ABB RobotStudio station: saddlewelding_2dofpositioner.rspag

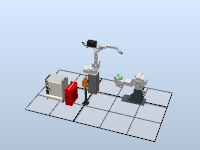
--- station ---
Station FInal3_1520_2dof (saved by RobotStudio 7.0.8743.626)
Controller Final3_1520_2dof, task T_ROB1: task frame (RAPID world) sits at (0, 0, 900) mm in the station
Controller Final3_1520_2dof
  mechanical unit ROB_1: IRB1520ID_4_150__02, 6 joints, base frame (0, 0, 0) mm
  mechanical unit STN1: IRBP_A250_D1000_M2009_REV1_01, 2 joints, base frame (0, 0, 0) mm
Layout (positions relative to the parent item):
  - IRB1520ID_4_150__02 [mechanism, from Robots\IRB1520ID_4_150_G_02.rslib] at (0, 0, 900) mm; joint values [0, 0, 0, 0, 0.5236, 0] (rad or m)
  - base900 [part, from Dissertation\base900.rslib]
  - IRBP_A250_D1000_M2009_REV1_01 [mechanism] at (1025, 0, 0) mm; joint values [0, 0] (rad or m)
      links: Base, Link1, Link2
  - Binzel_ID_22 [mechanism, from Tools\Binzel_ID_22.rslib] at (1056.21, 0, 2043) mm, rotated rx 180 ry 60 rz 180 deg
  - saddle_simple_tpipe [part] at (1025, 0, 940) mm, rotated rx 90 ry 0 rz 180 deg
  - Fronius_VR1500 [part, from Equipment\Fronius_VR1500.rslib] at (-224.71, 27.64, 723.67) mm
  - IRC5_Singel-Cabinet [part, from Equipment\IRC5_Singel-Cabinet.rslib] at (-1184.73, -1000, 100) mm, rotated rx 90 ry 0 rz 0 deg
  - Fronius_TPS4000_rev0 [part, from Equipment\Fronius_TPS4000.rslib] at (-575.52, -881.82, 0) mm, rotated rx 0 ry 0 rz 180 deg
  - torch_cleaner_binzel [graphiccomponentgroup, from Equipment\Torch Cleaner Binzel.rslib] at (0, -815.14, 0) mm
    - Body 1 [part, from Equipment\Torch Cleaner Binzel.rslib]
    - Body 2 [part, from Equipment\Torch Cleaner Binzel.rslib]
    - Body 3 [part, from Equipment\Torch Cleaner Binzel.rslib]
    - Body 4 [part, from Equipment\Torch Cleaner Binzel.rslib]
    - Body 5 [part, from Equipment\Torch Cleaner Binzel.rslib]
    - Body 6 [part, from Equipment\Torch Cleaner Binzel.rslib]
    - Body 7 [part, from Equipment\Torch Cleaner Binzel.rslib]
    - Body 8 [part, from Equipment\Torch Cleaner Binzel.rslib]
    - Body 9 [part, from Equipment\Torch Cleaner Binzel.rslib]
    - Body 10 [part, from Equipment\Torch Cleaner Binzel.rslib]
    - Body 11 [part, from Equipment\Torch Cleaner Binzel.rslib]
    - Body 12 [part, from Equipment\Torch Cleaner Binzel.rslib]
Attachment: Binzel_ID_22 is attached to IRB1520ID_4_150__02 / Link6
Attachment: saddle_simple_tpipe is attached to IRBP_A250_D1000_M2009_REV1_01 / Link2
Attachment: Fronius_VR1500 is attached to IRB1520ID_4_150__02 / Link3

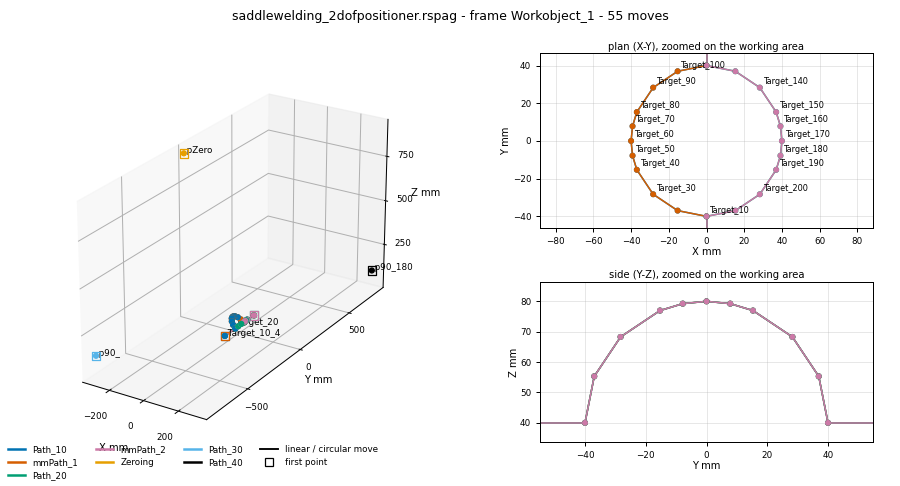
[picture p0: tool path of saddlewelding_2dofpositioner.rspag in frame Workobject_1, 55 of 55 moves have a stored position in this frame; points joined in program order, loops and branches not executed]
--- Backups/Final3_1520_2dof/RAPID/TASK1/PROGMOD/CalibData.mod ---
MODULE CalibData
	PERS tooldata tWeldGun:=[TRUE,[[49.841566361,0,372.194826196],[0.981627183,0,0.190808995,0]],[2,[0,0,100],[0,1,0,0],0,0,0]];
	TASK PERS wobjdata Workobject_1:=[FALSE,FALSE,"STN1",[[0,0,0],[1,0,0,0]],[[0,0,0],[1,0,0,0]]];
ENDMODULE

--- Backups/Final3_1520_2dof/RAPID/TASK1/PROGMOD/Module1.mod ---
MODULE Module1
	CONST robtarget Target_10_4:=[[0,-140,40],[0.653281482,-0.653281483,-0.27059805,-0.27059805],[0,0,0,0],[9E+09,9E+09,9E+09,9E+09,9E+09,9E+09]];
	CONST robtarget Target_10:=[[0,-40,40],[0.653281482,-0.653281483,-0.27059805,-0.27059805],[0,0,0,0],[9E+09,9E+09,9E+09,9E+09,9E+09,9E+09]];
	CONST robtarget Target_20:=[[-15.307337295,-36.9551813,55.307337295],[0.552498444,-0.741273461,-0.232815701,-0.301754825],[0,0,0,0],[9E+09,9E+09,9E+09,9E+09,9E+09,9E+09]];
	CONST robtarget Target_30:=[[-28.284271247,-28.284271247,68.284271247],[0.424708201,-0.820473238,-0.175919897,-0.339851143],[0,0,0,0],[9E+09,9E+09,9E+09,9E+09,9E+09,9E+09]];
	CONST robtarget Target_40:=[[-36.9551813,-15.307337295,76.9551813],[0.245447259,-0.877471606,-0.091255347,-0.401835396],[0,0,0,0],[9E+09,9E+09,9E+09,9E+09,9E+09,9E+09]];
	CONST robtarget Target_50:=[[-39.231411216,-7.803612881,79.231411216],[0.126767777,-0.911559828,-0.051100945,-0.387785125],[0,0,0,0],[9E+09,9E+09,9E+09,9E+09,9E+09,9E+09]];
	CONST robtarget Target_60:=[[-40,0,80],[0,0.923879533,0,0.382683432],[0,0,0,0],[9E+09,9E+09,9E+09,9E+09,9E+09,9E+09]];
	CONST robtarget Target_70:=[[-39.231411216,7.803612881,79.231411216],[0.126767777,0.911559828,-0.051100945,0.387785125],[0,0,0,0],[9E+09,9E+09,9E+09,9E+09,9E+09,9E+09]];
	CONST robtarget Target_80:=[[-36.9551813,15.307337295,76.9551813],[0.245447259,0.877471606,-0.091255347,0.401835396],[0,0,0,0],[9E+09,9E+09,9E+09,9E+09,9E+09,9E+09]];
	CONST robtarget Target_90:=[[-28.284271247,28.284271247,68.284271247],[0.424708201,0.820473238,-0.175919897,0.339851143],[0,0,0,0],[9E+09,9E+09,9E+09,9E+09,9E+09,9E+09]];
	CONST robtarget Target_100:=[[-15.307337295,36.9551813,55.307337295],[0.552498444,0.741273461,-0.232815702,0.301754825],[0,0,0,0],[9E+09,9E+09,9E+09,9E+09,9E+09,9E+09]];
	CONST robtarget Target_110:=[[0,40,40],[0.653281482,0.653281483,-0.27059805,0.27059805],[0,0,0,0],[9E+09,9E+09,9E+09,9E+09,9E+09,9E+09]];
	CONST robtarget Target_110_3:=[[0,140,40],[0.653281482,0.653281483,-0.27059805,0.27059805],[0,0,0,0],[9E+09,9E+09,9E+09,9E+09,9E+09,9E+09]];
	CONST robtarget pTarget_1:=[[0,-140,40],[0.653281482,-0.653281483,-0.27059805,-0.27059805],[-1,0,-1,0],[9E+09,-89.999998314,-0.000000734,9E+09,9E+09,9E+09]];
	CONST robtarget pTarget_2:=[[0,-40,40],[0.653281482,-0.653281483,-0.27059805,-0.27059805],[-1,0,-1,0],[9E+09,-89.802410692,4.557172082,9E+09,9E+09,9E+09]];
	CONST robtarget pTarget_3:=[[-15.307337295,-36.9551813,55.307337295],[0.552498444,-0.741273461,-0.232815701,-0.301754825],[-1,0,-1,0],[9E+09,-76.295977766,18.279214138,9E+09,9E+09,9E+09]];
	CONST robtarget pTarget_4:=[[-28.284271247,-28.284271247,68.284271247],[0.424708201,-0.820473238,-0.175919897,-0.339851143],[-1,0,-1,0],[9E+09,-61.411118651,37.565448127,9E+09,9E+09,9E+09]];
	CONST robtarget pTarget_5:=[[-36.9551813,-15.307337295,76.9551813],[0.245447259,-0.877471606,-0.091255347,-0.401835396],[-1,0,-2,0],[9E+09,-47.380570194,71.170137619,9E+09,9E+09,9E+09]];
	CONST robtarget pTarget_6:=[[-39.231411216,-7.803612881,79.231411216],[0.126767777,-0.911559828,-0.051100945,-0.387785125],[-1,0,-2,0],[9E+09,-36.088107809,97.239437874,9E+09,9E+09,9E+09]];
	CONST robtarget pTarget_7:=[[-40,0,80],[0,0.923879533,0,0.382683432],[-1,0,-2,0],[9E+09,-31.001963049,129.358833622,9E+09,9E+09,9E+09]];
	CONST robtarget pTarget_8:=[[-39.231411216,7.803612881,79.231411216],[0.126767777,0.911559828,-0.051100945,0.387785125],[-1,0,-2,0],[9E+09,-36.088107791,152.02186895,9E+09,9E+09,9E+09]];
	CONST robtarget pTarget_9:=[[-36.9551813,15.307337295,76.9551813],[0.245447259,0.877471606,-0.091255347,0.401835396],[-1,0,-2,0],[9E+09,-47.380570194,163.079129504,9E+09,9E+09,9E+09]];
	CONST robtarget pTarget_10:=[[-28.284271247,28.284271247,68.284271247],[0.424708201,0.820473238,-0.175919897,0.339851143],[-1,0,-2,0],[9E+09,-61.411118652,186.252573581,9E+09,9E+09,9E+09]];
	CONST robtarget pTarget_11:=[[-15.307337295,36.9551813,55.307337295],[0.552498444,0.741273461,-0.232815702,0.301754825],[-1,0,-2,0],[9E+09,-76.29597773,198.192760331,9E+09,9E+09,9E+09]];
	CONST robtarget pTarget_12:=[[0,40,40],[0.653281482,0.653281483,-0.27059805,0.27059805],[-1,0,-2,0],[9E+09,-89.802410695,207.373271387,9E+09,9E+09,9E+09]];
	CONST robtarget pTarget_13:=[[0,140,40],[0.653281482,0.653281483,-0.27059805,0.27059805],[-1,0,-2,0],[9E+09,-89.999998314,199.574847217,9E+09,9E+09,9E+09]];
	CONST robtarget Target_120_2:=[[0,140,40],[0.27059805,0.27059805,-0.653281483,0.653281482],[0,0,0,0],[9E+09,9E+09,9E+09,9E+09,9E+09,9E+09]];
	CONST robtarget Target_120:=[[0,40,40],[0.27059805,0.27059805,-0.653281483,0.653281482],[0,0,0,0],[9E+09,9E+09,9E+09,9E+09,9E+09,9E+09]];
	CONST robtarget Target_130:=[[15.307337295,36.9551813,55.307337295],[0.301754825,0.232815701,-0.741273461,0.552498444],[0,0,0,0],[9E+09,9E+09,9E+09,9E+09,9E+09,9E+09]];
	CONST robtarget Target_140:=[[28.284271247,28.284271247,68.284271247],[0.339851143,0.175919897,-0.820473239,0.4247082],[0,0,0,0],[9E+09,9E+09,9E+09,9E+09,9E+09,9E+09]];
	CONST robtarget Target_150:=[[36.9551813,15.307337295,76.9551813],[0.401835396,0.091255347,-0.877471606,0.245447259],[0,0,0,0],[9E+09,9E+09,9E+09,9E+09,9E+09,9E+09]];
	CONST robtarget Target_160:=[[39.231411216,7.803612881,79.231411216],[0.387785125,0.051100945,-0.911559828,0.126767777],[0,0,0,0],[9E+09,9E+09,9E+09,9E+09,9E+09,9E+09]];
	CONST robtarget Target_170:=[[40,0,80],[0.382683432,0,-0.923879533,0],[0,0,0,0],[9E+09,9E+09,9E+09,9E+09,9E+09,9E+09]];
	CONST robtarget Target_180:=[[39.231411216,-7.803612881,79.231411216],[0.387785125,-0.051100945,-0.911559828,-0.126767777],[0,0,0,0],[9E+09,9E+09,9E+09,9E+09,9E+09,9E+09]];
	CONST robtarget Target_190:=[[36.9551813,-15.307337295,76.9551813],[0.401835396,-0.091255347,-0.877471606,-0.245447259],[0,0,0,0],[9E+09,9E+09,9E+09,9E+09,9E+09,9E+09]];
	CONST robtarget Target_200:=[[28.284271247,-28.284271247,68.284271247],[0.339851143,-0.175919897,-0.820473239,-0.4247082],[0,0,0,0],[9E+09,9E+09,9E+09,9E+09,9E+09,9E+09]];
	CONST robtarget Target_210:=[[15.307337295,-36.9551813,55.307337295],[0.301754825,-0.232815702,-0.741273461,-0.552498444],[0,0,0,0],[9E+09,9E+09,9E+09,9E+09,9E+09,9E+09]];
	CONST robtarget Target_220:=[[0,-40,40],[0.27059805,-0.27059805,-0.653281483,-0.653281482],[0,0,0,0],[9E+09,9E+09,9E+09,9E+09,9E+09,9E+09]];
	CONST robtarget Target_220_2:=[[0,-140,40],[0.27059805,-0.27059805,-0.653281483,-0.653281482],[0,0,0,0],[9E+09,9E+09,9E+09,9E+09,9E+09,9E+09]];
	CONST robtarget pTarget_14:=[[0,140,40],[0.27059805,0.27059805,-0.653281483,0.653281482],[-1,0,-1,0],[9E+09,-89.999998314,179.999999266,9E+09,9E+09,9E+09]];
	CONST robtarget pTarget_15:=[[0,40,40],[0.27059805,0.27059805,-0.653281483,0.653281482],[-1,0,-1,0],[9E+09,-89.802410692,184.557172082,9E+09,9E+09,9E+09]];
	CONST robtarget pTarget_16:=[[15.307337295,36.9551813,55.307337295],[0.301754825,0.232815701,-0.741273461,0.552498444],[-1,0,-1,0],[9E+09,-76.295977766,198.279214138,9E+09,9E+09,9E+09]];
	CONST robtarget pTarget_17:=[[28.284271247,28.284271247,68.284271247],[0.339851143,0.175919897,-0.820473239,0.4247082],[-1,0,-1,0],[9E+09,-61.411118499,217.565448249,9E+09,9E+09,9E+09]];
	CONST robtarget pTarget_18:=[[36.9551813,15.307337295,76.9551813],[0.401835396,0.091255347,-0.877471606,0.245447259],[-1,0,-2,0],[9E+09,-47.380570194,251.170137619,9E+09,9E+09,9E+09]];
	CONST robtarget pTarget_19:=[[39.231411216,7.803612881,79.231411216],[0.387785125,0.051100945,-0.911559828,0.126767777],[-1,0,-2,0],[9E+09,-36.088107809,277.239437874,9E+09,9E+09,9E+09]];
	CONST robtarget pTarget_20:=[[40,0,80],[0.382683432,0,-0.923879533,0],[-1,0,-2,0],[9E+09,-31.001963049,309.358833622,9E+09,9E+09,9E+09]];
	CONST robtarget pTarget_21:=[[39.231411216,-7.803612881,79.231411216],[0.387785125,-0.051100945,-0.911559828,-0.126767777],[-1,0,-2,0],[9E+09,-36.088107791,332.02186895,9E+09,9E+09,9E+09]];
	CONST robtarget pTarget_22:=[[36.9551813,-15.307337295,76.9551813],[0.401835396,-0.091255347,-0.877471606,-0.245447259],[-1,0,-2,0],[9E+09,-47.380570194,343.079129504,9E+09,9E+09,9E+09]];
	CONST robtarget pTarget_23:=[[28.284271247,-28.284271247,68.284271247],[0.339851143,-0.175919897,-0.820473239,-0.4247082],[-1,0,-2,0],[9E+09,-61.4111185,366.252573561,9E+09,9E+09,9E+09]];
	CONST robtarget pTarget_24:=[[15.307337295,-36.9551813,55.307337295],[0.301754825,-0.232815702,-0.741273461,-0.552498444],[-1,0,-2,0],[9E+09,-76.29597773,378.192760331,9E+09,9E+09,9E+09]];
	CONST robtarget pTarget_25:=[[0,-40,40],[0.27059805,-0.27059805,-0.653281483,-0.653281482],[-1,0,-2,0],[9E+09,-89.802410695,387.373271387,9E+09,9E+09,9E+09]];
	CONST robtarget pTarget_26:=[[0,-140,40],[0.27059805,-0.27059805,-0.653281483,-0.653281482],[-1,0,-2,0],[9E+09,-89.999998314,379.574847217,9E+09,9E+09,9E+09]];
	CONST robtarget pZero:=[[-328.614472219,0,913.738524269],[0,0.945518575,0,-0.325568155],[0,0,0,0],[9E+09,0,0,9E+09,9E+09,9E+09]];
	CONST robtarget p90_:=[[-328.614472219,-793.738524269,120.000029927],[0.668582584,-0.668582609,-0.230211446,0.230211454],[0,0,0,0],[9E+09,-89.99999784,0,9E+09,9E+09,9E+09]];
	CONST robtarget p90_180:=[[328.614472219,793.738524269,120.000029927],[0.230211454,-0.230211446,0.668582609,-0.668582584],[0,0,0,0],[9E+09,-89.99999784,180,9E+09,9E+09,9E+09]];
    !***********************************************************
    !
    ! Module:  Module1
    !
    ! Description:
    !   <Insert description here>
    !
    ! Author: firmi
    !
    ! Version: 1.0
    !
    !***********************************************************


    !***********************************************************
    !
    ! Procedure main
    !
    !   This is the entry point of your program
    !
    !***********************************************************
    PROC main()
        !Add your code here
        DeactUnit STN1;
        ActUnit STN1;
        Zeroing;
        Path_30;
        mmPath_1;
        Path_40;
        mmPath_2;
        Zeroing;
        DeactUnit STN1;


    ENDPROC
	PROC Path_10()
	    MoveL Target_10_4,v50,z0,tWeldGun\WObj:=Workobject_1;
	    MoveL Target_10,v50,z0,tWeldGun\WObj:=Workobject_1;
	    MoveL Target_20,v50,z0,tWeldGun\WObj:=Workobject_1;
	    MoveL Target_30,v50,z0,tWeldGun\WObj:=Workobject_1;
	    MoveL Target_40,v50,z0,tWeldGun\WObj:=Workobject_1;
	    MoveL Target_50,v50,z0,tWeldGun\WObj:=Workobject_1;
	    MoveL Target_60,v50,z0,tWeldGun\WObj:=Workobject_1;
	    MoveL Target_70,v50,z0,tWeldGun\WObj:=Workobject_1;
	    MoveL Target_80,v50,z0,tWeldGun\WObj:=Workobject_1;
	    MoveL Target_90,v50,z0,tWeldGun\WObj:=Workobject_1;
	    MoveL Target_100,v50,z0,tWeldGun\WObj:=Workobject_1;
	    MoveL Target_110,v50,z0,tWeldGun\WObj:=Workobject_1;
	    MoveL Target_110_3,v50,z0,tWeldGun\WObj:=Workobject_1;
	ENDPROC
	PROC mmPath_1()
	    MoveL pTarget_1,v50,z0,tWeldGun\WObj:=Workobject_1;
	    MoveL pTarget_2,v50,z0,tWeldGun\WObj:=Workobject_1;
	    MoveL pTarget_3,v50,z0,tWeldGun\WObj:=Workobject_1;
	    MoveL pTarget_4,v50,z0,tWeldGun\WObj:=Workobject_1;
	    MoveL pTarget_5,v50,z0,tWeldGun\WObj:=Workobject_1;
	    MoveL pTarget_6,v50,z0,tWeldGun\WObj:=Workobject_1;
	    MoveL pTarget_7,v50,z0,tWeldGun\WObj:=Workobject_1;
	    MoveL pTarget_8,v50,z0,tWeldGun\WObj:=Workobject_1;
	    MoveL pTarget_9,v50,z0,tWeldGun\WObj:=Workobject_1;
	    MoveL pTarget_10,v50,z0,tWeldGun\WObj:=Workobject_1;
	    MoveL pTarget_11,v50,z0,tWeldGun\WObj:=Workobject_1;
	    MoveL pTarget_12,v50,z0,tWeldGun\WObj:=Workobject_1;
	    MoveL pTarget_13,v50,z0,tWeldGun\WObj:=Workobject_1;
	ENDPROC
	PROC Path_20()
	    MoveL Target_120_2,v50,z0,tWeldGun\WObj:=Workobject_1;
	    MoveL Target_120,v50,z0,tWeldGun\WObj:=Workobject_1;
	    MoveL Target_130,v50,z0,tWeldGun\WObj:=Workobject_1;
	    MoveL Target_140,v50,z0,tWeldGun\WObj:=Workobject_1;
	    MoveL Target_150,v50,z0,tWeldGun\WObj:=Workobject_1;
	    MoveL Target_160,v50,z0,tWeldGun\WObj:=Workobject_1;
	    MoveL Target_170,v50,z0,tWeldGun\WObj:=Workobject_1;
	    MoveL Target_180,v50,z0,tWeldGun\WObj:=Workobject_1;
	    MoveL Target_190,v50,z0,tWeldGun\WObj:=Workobject_1;
	    MoveL Target_200,v50,z0,tWeldGun\WObj:=Workobject_1;
	    MoveL Target_210,v50,z0,tWeldGun\WObj:=Workobject_1;
	    MoveL Target_220,v50,z0,tWeldGun\WObj:=Workobject_1;
	    MoveL Target_220_2,v50,z0,tWeldGun\WObj:=Workobject_1;
	ENDPROC
	PROC mmPath_2()
	    MoveL pTarget_14,v50,z0,tWeldGun\WObj:=Workobject_1;
	    MoveL pTarget_15,v50,z0,tWeldGun\WObj:=Workobject_1;
	    MoveL pTarget_16,v50,z0,tWeldGun\WObj:=Workobject_1;
	    MoveL pTarget_17,v50,z0,tWeldGun\WObj:=Workobject_1;
	    MoveL pTarget_18,v50,z0,tWeldGun\WObj:=Workobject_1;
	    MoveL pTarget_19,v50,z0,tWeldGun\WObj:=Workobject_1;
	    MoveL pTarget_20,v50,z0,tWeldGun\WObj:=Workobject_1;
	    MoveL pTarget_21,v50,z0,tWeldGun\WObj:=Workobject_1;
	    MoveL pTarget_22,v50,z0,tWeldGun\WObj:=Workobject_1;
	    MoveL pTarget_23,v50,z0,tWeldGun\WObj:=Workobject_1;
	    MoveL pTarget_24,v50,z0,tWeldGun\WObj:=Workobject_1;
	    MoveL pTarget_25,v50,z0,tWeldGun\WObj:=Workobject_1;
	    MoveL pTarget_26,v50,z0,tWeldGun\WObj:=Workobject_1;
	ENDPROC
	PROC Zeroing()
	    MoveJ pZero,v50,z0,tWeldGun\WObj:=Workobject_1;
	ENDPROC
	PROC Path_30()
	    MoveL p90_,v50,z0,tWeldGun\WObj:=Workobject_1;
	ENDPROC
	PROC Path_40()
	    MoveL p90_180,v50,z0,tWeldGun\WObj:=Workobject_1;
	ENDPROC
ENDMODULE

--- Backups/Final3_1520_2dof/SYSPAR/EIO.cfg ---
EIO:CFG_1.0:6:1::
#
LOCAL_DEVICE:

      -Name "DRVIO_1" -Network "Local" -StateWhenStartup "Deactivated"\
      -TrustLevel "DRVIO_TRUSTLEVEL"
#
EIO_CROSS:

      -Name "Cross_doACT_K1" -Res "doACT_K1" -Act1 "soACT_STN1"

      -Name "Cross_doACT_K3" -Res "doACT_K3" -Act1 "soACT_STN1"

      -Name "Cross_siSTN1_ACT" -Res "siSTN1_ACT" -Act1 "diK1_ACT" -Oper1 "AND"\
      -Act2 "diK3_ACT"

      -Name "Cross_doACT_K11" -Res "doACT_K11" -Act1 "doACT_K13"
#
EIO_DEVICE_TRUSTLEVEL:

      -Name "DRVIO_TRUSTLEVEL" -ActionWhenLost "NONE" -ReportWhenLost "NONE"\
      -ReportWhenReconnected "NONE"
#
EIO_SIGNAL:

      -Name "doACT_K1" -SignalType "DO" -Device "DRVIO_1" -DeviceMap "0"

      -Name "doACT_K3" -SignalType "DO" -Device "DRVIO_1" -DeviceMap "2"

      -Name "doACT_K11" -SignalType "DO" -Device "DRVIO_1" -DeviceMap "5"

      -Name "doACT_K13" -SignalType "DO" -Device "DRVIO_1" -DeviceMap "7"

      -Name "diK1_ACT" -SignalType "DI" -Device "DRVIO_1" -DeviceMap "0"\
      -FiltPas 50 -FiltAct 50

      -Name "diK3_ACT" -SignalType "DI" -Device "DRVIO_1" -DeviceMap "2"\
      -FiltPas 50 -FiltAct 50

      -Name "soACT_STN1" -SignalType "DO" -DeviceMap "0"

      -Name "siSTN1_ACT" -SignalType "DI" -DeviceMap "0"
